# EPICS substitutions: db/MicroEpsilon/ecmcCapaNCDT6200.substitutions
file "ecmc_analogInputFloat-chX.template"
{
  pattern { CH_ID,  KEY,   EGU,  PREC,  suffix    }
          { 01,     "Enc", "um", 1,     "-PosAct"  }
          { 02,     "Enc", "um", 1,     "-PosAct"  }
          { 03,     "Enc", "um", 1,     "-PosAct"  }
          { 04,     "Enc", "um", 1,     "-PosAct"  }
}
